Universal Robots PolyScope program: cottonDisplay.urp

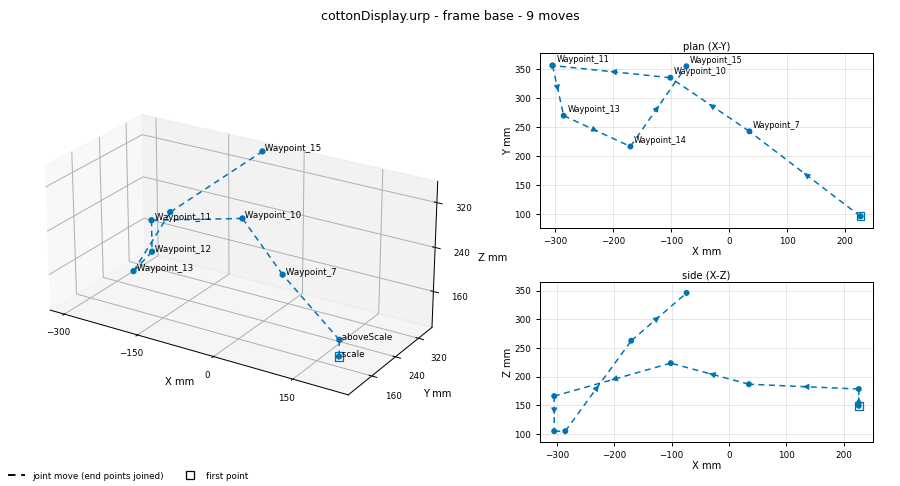
[picture p0: tool path of cottonDisplay.urp in frame base, 9 of 10 moves have a stored position in this frame; points joined in program order, loops and branches not executed]
Program cottonDisplay (installation=default directory=/programs/DavidMelin createdIn=5.12.4.1101661 lastSavedIn=5.12.4.1101661 robotSerialNumber=20225502378)
Calibrated DH parameters: a=[0.00022, -0.425328, -0.389701, 0.000059, 0.000065, 0]; d=[0.162608, 0.803456, 9.992211, -10.662202, 0.099702, 0.099559]; alpha=[1.570756, 0.001543, 0.004316, 1.570651, -1.570122, 0]; deltaTheta=[0, 0.002917, 0.116094, -0.119008, 0, -0.000001]
Robot Program (runOnlyOnce=true)
  URCap Gripper (Robotiq_Grippers, Robotiq Inc.) dataModel(position=0.0, force=0.0, speed=0.0, positionInDouble=0.0, forceInDouble=0.0, speedInDouble=0.0, slaveIds=[9], blocking=true)
  MoveJ speed 60 deg/s, acceleration 80 deg/s^2 (useActiveTCP=true) feature=Base
    Waypoint scale: TCP in base x=226.483 y=96.053 z=149.343 mm, rx=-1.5818 ry=-0.3301 rz=0.3435 rad; joints [31.27, -97.11, -141.687, -135.565, -172.89, 166.689] deg
  URCap Gripper (Robotiq_Grippers, Robotiq Inc.) dataModel(position=95.09803921568627, force=0.0, speed=0.0, positionInDouble=95.09803921568627, forceInDouble=0.0, speedInDouble=0.0, slaveIds=[9], blocking=true)
  MoveJ speed 60 deg/s, acceleration 80 deg/s^2 (useActiveTCP=true) feature=Base
    Waypoint aboveScale: TCP in base x=226.497 y=96.066 z=178.622 mm, rx=-1.5818 ry=-0.3301 rz=0.3435 rad; joints [31.277, -91.949, -140.091, -142.239, -172.906, 166.771] deg
    Waypoint Waypoint_7: TCP in base x=34.857 y=242.691 z=186.982 mm, rx=-1.2726 ry=-1.1534 rz=1.097 rad; joints [90.147, -89.974, -140.099, -142.249, -172.955, 166.769] deg
    Waypoint Waypoint_10: TCP in base x=-101.456 y=335.252 z=223.697 mm, rx=-1.2953 ry=-1.0334 rz=1.1569 rad; joints [115.421, -89.57, -133.643, -132.861, -145.414, 187.147] deg
    Waypoint Waypoint_11: TCP in base x=-304.815 y=356.228 z=166.249 mm, rx=-1.5536 ry=-0.0689 rz=0.1544 rad; joints [158.685, -106.013, -125.631, -126.585, -29.374, 181.619] deg
    Waypoint Waypoint_12: TCP in base x=-304.823 y=356.244 z=105.048 mm, rx=-1.5536 ry=-0.0688 rz=0.1545 rad; joints [158.675, -114.599, -127.491, -116.094, -29.35, 181.573] deg
  URCap Gripper (Robotiq_Grippers, Robotiq Inc.) dataModel(position=0.0, force=0.0, speed=0.0, positionInDouble=0.0, forceInDouble=0.0, speedInDouble=0.0, slaveIds=[9], blocking=true)
  MoveJ speed 60 deg/s, acceleration 80 deg/s^2 (useActiveTCP=true) feature=Base
    Waypoint Waypoint_13: TCP in base x=-285.543 y=269.692 z=105.058 mm, rx=-1.5536 ry=-0.0689 rz=0.1545 rad; joints [172.49, -108.656, -139.043, -108.935, -15.541, 179.865] deg
    Waypoint Waypoint_14: TCP in base x=-170.402 y=216.56 z=262.874 mm, rx=-1.6767 ry=1.1987 rz=0.1014 rad; joints [178.185, -59.547, -143.413, -109.321, 39.618, 179.866] deg
    Waypoint Waypoint_15: TCP in base x=-73.88 y=354.943 z=346.223 mm, rx=-2.7227 ry=0.6943 rz=0.1377 rad; joints [126.714, -68.027, -133.751, -51.903, 79.219, 63.781] deg
    Waypoint Waypoint (Variable): variable=cotonHomePos
